PROGRAM MAIN

VAR
	fbSafetyX : fb_safety;
	fbSafetyY : fb_safety;
	fbSystemBufferX : fb_StatusBuffer;
	fbSystemBufferY : fb_StatusBuffer;
	fbMovementControllerX : fb_MovementController;
	fbMovementControllerY : fb_MovementController;
	fbBiaxialCoordinator : fb_BiaxialCoordinator;
	fbStatusPublisherX : fb_AxisStatusPublisher;
	fbStatusPublisherY : fb_AxisStatusPublisher;
	
	// DUTs import
	stMoveCommandX : ST_MoveCommand;
	stMoveCommandY : ST_MoveCommand;

	stSystemStatusX : ST_SystemStatus;
	stSystemStatusY : ST_SystemStatus;

	stSettingsX : ST_Settings;
	stSettingsY : ST_Settings;

	// IO Links
    nRawTenzoX AT %I* : DINT;
	nRawTenzoY AT %I* : DINT;

	nEndStopLx AT %I* : BOOL;
	nEndStopHx AT %I* : BOOL;

	nEndStopLy AT %I* : BOOL;
	nEndStopHy AT %I* : BOOL;

	// Normalized physical limits: TRUE means that the switch is pressed.
	bEndStopLxActive : BOOL;
	bEndStopHxActive : BOOL;
	bEndStopLyActive : BOOL;
	bEndStopHyActive : BOOL;

	// PLC-owned synchronized start request
	bStartBiaxialTest : BOOL; // ADS one-shot after both axis commands are prepared

	// Persistent-axis checkpoint diagnostics. A successful checkpoint creates
	// an up-to-date Port_851.bootdata file before controller power is removed.
	bPersistentPositionSaved : BOOL;
	bPersistentPositionSaveBusy : BOOL;
	bPersistentPositionSaveError : BOOL;
	nPersistentPositionSaveErrorID : UDINT;
	nPersistentPositionCheckpointCounter : UDINT;

	fbWritePersistentData : FB_WritePersistentData;
	fbPersistentPositionSettle : TON;
	ftPowerRequestX : F_TRIG;
	ftPowerRequestY : F_TRIG;
	rtPersistentValidX : R_TRIG;
	rtPersistentValidY : R_TRIG;
	bPersistentInitialCheckpoint : BOOL := TRUE;
	bPersistentCheckpointPending : BOOL;
	bPersistentCheckpointInFlight : BOOL;
	bPersistentCheckpointStart : BOOL;
	bPersistentSafeToWrite : BOOL;
	nPersistentCheckpointRequestGeneration : UDINT;
	nPersistentCheckpointStartedGeneration : UDINT;
	nPersistentCheckpointCompletedGeneration : UDINT;
	fCheckpointPositionX : LREAL;
	fCheckpointPositionY : LREAL;
	bCheckpointValidX : BOOL;
	bCheckpointValidY : BOOL;

END_VAR

VAR_TEMP
	bBiaxialAxesReady : BOOL;
	bBiaxialCommonAbortRequest : BOOL;
	bRestoreReferenceX : BOOL;
	bRestoreReferenceY : BOOL;
END_VAR

////////////////////////////////
//////////   safety   //////////
////////////////////////////////

// Refresh NC status before making any safety or motion decision
GVL_Axis.xAxis.ReadStatus();
GVL_Axis.yAxis.ReadStatus();

// Requesting a physical home deliberately invalidates the old retained
// coordinate. Only a successfully referenced axis will make it valid again.
IF stMoveCommandX.bHome THEN
	GVL_Persistent.bLastPositionValidX := FALSE;
END_IF
IF stMoveCommandY.bHome THEN
	GVL_Persistent.bLastPositionValidY := FALSE;
END_IF

// On the first powered scan after a PLC/NC restart, statically restore each
// incremental axis to its last persistent coordinate. MC_Direct performs no
// motor movement. A normal reference-cam home always takes priority.
bRestoreReferenceX :=
	GVL_Persistent.bLastPositionValidX AND
	NOT GVL_Axis.xAxis.Status.Homed AND
	NOT fbSafetyX.bReferenceRestoreDone;
bRestoreReferenceY :=
	GVL_Persistent.bLastPositionValidY AND
	NOT GVL_Axis.yAxis.Status.Homed AND
	NOT fbSafetyY.bReferenceRestoreDone;

// Normalize the active-low physical switches
bEndStopLxActive := NOT nEndStopLx;
bEndStopHxActive := NOT nEndStopHx;
bEndStopLyActive := NOT nEndStopLy;
bEndStopHyActive := NOT nEndStopHy;

fbSafetyX(
    stAxis := GVL_Axis.xAxis,
    bPower := stMoveCommandX.bPower,
    bReset := stMoveCommandX.bReset,
    bHalt := stMoveCommandX.bHalt OR fbMovementControllerX.stateHalt,
    bHome := stMoveCommandX.bHome,
	bRestoreReference := bRestoreReferenceX,
	fRestoreReferencePosition := GVL_Persistent.fLastPositionX,
    bEndStopL := bEndStopLxActive,
	bEndStopH := bEndStopHxActive,
	bExternalBusy := fbMovementControllerX.bBusy OR stSystemStatusX.bTarWorking
);

fbSafetyY(
    stAxis := GVL_Axis.yAxis,
    bPower := stMoveCommandY.bPower,
    bReset := stMoveCommandY.bReset,
    bHalt := stMoveCommandY.bHalt OR fbMovementControllerY.stateHalt,
    bHome := stMoveCommandY.bHome,
	bRestoreReference := bRestoreReferenceY,
	fRestoreReferencePosition := GVL_Persistent.fLastPositionY,
    bEndStopL := bEndStopLyActive,
	bEndStopH := bEndStopHyActive,
	bExternalBusy := fbMovementControllerY.bBusy OR stSystemStatusY.bTarWorking
);

////////////////////////////////
////////// Update data /////////
////////////////////////////////

fbSystemBufferX(
	stSystemStatus:= stSystemStatusX,
	bBlockTar:= fbMovementControllerX.bBusy OR fbSafetyX.bHoming OR
		NOT fbSafetyX.bHomed,
	nRawTenzo:= -nRawTenzoX,
	fTenzoCons:=stSettingsX.fTenzoCons,
	fTenzoOffset:= stSettingsX.fTenzoOffset,
	bStartTar:= stMoveCommandX.bStartTar,
	fActPosition:= GVL_Axis.xAxis.NcToPlc.ActPos);
	
fbSystemBufferY(
	stSystemStatus:= stSystemStatusY,
	bBlockTar:= fbMovementControllerY.bBusy OR fbSafetyY.bHoming OR
		NOT fbSafetyY.bHomed,
	nRawTenzo:= nRawTenzoY,
	fTenzoCons:=stSettingsY.fTenzoCons,
	fTenzoOffset:= stSettingsY.fTenzoOffset,
	bStartTar:= stMoveCommandY.bStartTar,
	fActPosition:= GVL_Axis.yAxis.NcToPlc.ActPos);

/////////////////////////////////////
////////// Main Move Logic //////////
/////////////////////////////////////

// A shared request starts both axes in one PLC scan. Single-axis tests keep
// using their individual bExecute fields and never enable synchronization.
bBiaxialAxesReady :=
	NOT fbMovementControllerX.bBusy AND
	NOT fbMovementControllerY.bBusy AND
	NOT fbMovementControllerX.bError AND
	NOT fbMovementControllerY.bError AND
	NOT fbSafetyX.bError AND NOT fbSafetyY.bError AND
	NOT fbSafetyX.bHoming AND NOT fbSafetyY.bHoming AND
	fbSafetyX.bHomed AND fbSafetyY.bHomed AND
	NOT stSystemStatusX.bTarWorking AND
	NOT stSystemStatusY.bTarWorking AND
	fbSafetyX.bPowerStatus AND fbSafetyY.bPowerStatus;

// Ignore ProtectiveStop when it was produced by the controller's own
// controlled halt. Operator, end-stop and independent safety stops abort both
// axes; an overforce relief request aborts only the synchronized peer.
bBiaxialCommonAbortRequest :=
	fbMovementControllerX.bError OR fbMovementControllerY.bError OR
	fbSafetyX.bError OR fbSafetyY.bError OR
	(fbSafetyX.bProtectiveStop AND
	 NOT fbMovementControllerX.stateHalt) OR
	(fbSafetyY.bProtectiveStop AND
	 NOT fbMovementControllerY.stateHalt) OR
	(bEndStopLxActive AND GVL_Axis.xAxis.Status.NegativeDirection) OR
	(bEndStopHxActive AND GVL_Axis.xAxis.Status.PositiveDirection) OR
	(bEndStopLyActive AND GVL_Axis.yAxis.Status.NegativeDirection) OR
	(bEndStopHyActive AND GVL_Axis.yAxis.Status.PositiveDirection) OR
	stMoveCommandX.bHalt OR stMoveCommandY.bHalt;

fbBiaxialCoordinator(
	bStartRequest := bStartBiaxialTest,
	bResetRequest := stMoveCommandX.bReset OR stMoveCommandY.bReset,
	bAxesReady := bBiaxialAxesReady,
	bCommonAbortRequest := bBiaxialCommonAbortRequest,
	bBusyX := fbMovementControllerX.bBusy,
	bBusyY := fbMovementControllerY.bBusy,
	bSavedPositionValidX := fbMovementControllerX.bSavedPositionValid,
	bSavedPositionValidY := fbMovementControllerY.bSavedPositionValid,
	nSyncPointX := fbMovementControllerX.nSyncPoint,
	nSyncPointY := fbMovementControllerY.nSyncPoint,
	nSyncCycleX := fbMovementControllerX.nSyncCycle,
	nSyncCycleY := fbMovementControllerY.nSyncCycle,
	bPeerAbortRequestX := fbMovementControllerX.bPeerAbortRequest,
	bPeerAbortRequestY := fbMovementControllerY.bPeerAbortRequest,
	stCommandX := stMoveCommandX,
	stCommandY := stMoveCommandY);

IF bStartBiaxialTest THEN
	bStartBiaxialTest := FALSE;
END_IF

IF fbBiaxialCoordinator.bStartBoth THEN
	stMoveCommandX.bExecute := TRUE;
	stMoveCommandY.bExecute := TRUE;
END_IF

fbMovementControllerX(
	Axis := GVL_Axis.xAxis,
	stMoveCommand := stMoveCommandX,
	stSettings := stSettingsX,
	fActPosition := GVL_Axis.xAxis.NcToPlc.ActPos,
    bPowerState := fbSafetyX.bPowerStatus,
	bHaltDone := fbSafetyX.bHaltDone,
	bAxisStopped := fbSafetyX.bStopped,
	bSafetyError := fbSafetyX.bError,
	bProtectiveStop := fbSafetyX.bProtectiveStop,
	bExternalBusy := fbSafetyX.bHoming OR
		NOT fbSafetyX.bHomed OR stSystemStatusX.bTarWorking,
	bReferenceValid := fbSafetyX.bHomed,
	bInvalidateSavedPosition := stMoveCommandX.bHome,
	bSyncEnabled := fbBiaxialCoordinator.bSyncActive,
	bSyncRelease := fbBiaxialCoordinator.bSyncRelease,
	bSyncAbort := fbBiaxialCoordinator.bAbortX,
	bSyncSingleComplete := fbBiaxialCoordinator.bSingleCompleteX,
    fForce := stSystemStatusX.fTenzoBuffer[stSystemStatusX.nBufferHead]);

fbMovementControllerY(
	Axis := GVL_Axis.yAxis,
	stMoveCommand := stMoveCommandY,
	stSettings := stSettingsY,
	fActPosition := GVL_Axis.yAxis.NcToPlc.ActPos,
    bPowerState := fbSafetyY.bPowerStatus,
	bHaltDone := fbSafetyY.bHaltDone,
	bAxisStopped := fbSafetyY.bStopped,
	bSafetyError := fbSafetyY.bError,
	bProtectiveStop := fbSafetyY.bProtectiveStop,
	bExternalBusy := fbSafetyY.bHoming OR
		NOT fbSafetyY.bHomed OR stSystemStatusY.bTarWorking,
	bReferenceValid := fbSafetyY.bHomed,
	bInvalidateSavedPosition := stMoveCommandY.bHome,
	bSyncEnabled := fbBiaxialCoordinator.bSyncActive,
	bSyncRelease := fbBiaxialCoordinator.bSyncRelease,
	bSyncAbort := fbBiaxialCoordinator.bAbortY,
	bSyncSingleComplete := fbBiaxialCoordinator.bSingleCompleteY,
	fForce := stSystemStatusY.fTenzoBuffer[stSystemStatusY.nBufferHead]);

///////////////////////////////////////////////////
////// ADS status contract for each axis //////////
///////////////////////////////////////////////////

fbStatusPublisherX(
	fActPosition := GVL_Axis.xAxis.NcToPlc.ActPos,
	bPowerStatus := fbSafetyX.bPowerStatus,
	bHoming := fbSafetyX.bHoming,
	bHomed := fbSafetyX.bHomed,
	bStopped := fbSafetyX.bStopped,
	bProtectiveStop := fbSafetyX.bProtectiveStop,
	bControllerHalt := fbMovementControllerX.stateHalt,
	bSafetyError := fbSafetyX.bError,
	nSafetyErrorCode := fbSafetyX.nErrorCode,
	nSafetyAxisErrorID := fbSafetyX.nAxisErrorID,
	bMovementBusy := fbMovementControllerX.bBusy,
	bMovementError := fbMovementControllerX.bError,
	nMovementStatus := fbMovementControllerX.nSystemStatus,
	nMovementErrorCode := fbMovementControllerX.nErrorCode,
	nMovementAxisErrorID := fbMovementControllerX.nAxisErrorID,
	nOperationCounter := fbMovementControllerX.nOperationCounter,
	bSavedPositionValid := fbMovementControllerX.bSavedPositionValid,
	bStartError := fbBiaxialCoordinator.bStartError,
	nStartErrorCode := fbBiaxialCoordinator.nStartErrorCode,
	stSystemStatus := stSystemStatusX);

fbStatusPublisherY(
	fActPosition := GVL_Axis.yAxis.NcToPlc.ActPos,
	bPowerStatus := fbSafetyY.bPowerStatus,
	bHoming := fbSafetyY.bHoming,
	bHomed := fbSafetyY.bHomed,
	bStopped := fbSafetyY.bStopped,
	bProtectiveStop := fbSafetyY.bProtectiveStop,
	bControllerHalt := fbMovementControllerY.stateHalt,
	bSafetyError := fbSafetyY.bError,
	nSafetyErrorCode := fbSafetyY.nErrorCode,
	nSafetyAxisErrorID := fbSafetyY.nAxisErrorID,
	bMovementBusy := fbMovementControllerY.bBusy,
	bMovementError := fbMovementControllerY.bError,
	nMovementStatus := fbMovementControllerY.nSystemStatus,
	nMovementErrorCode := fbMovementControllerY.nErrorCode,
	nMovementAxisErrorID := fbMovementControllerY.nAxisErrorID,
	nOperationCounter := fbMovementControllerY.nOperationCounter,
	bSavedPositionValid := fbMovementControllerY.bSavedPositionValid,
	bStartError := fbBiaxialCoordinator.bStartError,
	nStartErrorCode := fbBiaxialCoordinator.nStartErrorCode,
	stSystemStatus := stSystemStatusY);

// Track the last valid coordinate continuously in persistent PLC memory.
// Values are never replaced while an axis is unreferenced, homing, or in an
// NC error, so startup cannot accidentally retain the raw zero coordinate.
IF fbSafetyX.bHomed AND NOT fbSafetyX.bHoming AND
	NOT GVL_Axis.xAxis.Status.Error AND
	(GVL_Axis.xAxis.NcToPlc.ActPos =
		GVL_Axis.xAxis.NcToPlc.ActPos) AND
	ABS(GVL_Axis.xAxis.NcToPlc.ActPos) < 1.0E300 THEN
	GVL_Persistent.fLastPositionX :=
		GVL_Axis.xAxis.NcToPlc.ActPos;
	GVL_Persistent.bLastPositionValidX := TRUE;
END_IF

IF fbSafetyY.bHomed AND NOT fbSafetyY.bHoming AND
	NOT GVL_Axis.yAxis.Status.Error AND
	(GVL_Axis.yAxis.NcToPlc.ActPos =
		GVL_Axis.yAxis.NcToPlc.ActPos) AND
	ABS(GVL_Axis.yAxis.NcToPlc.ActPos) < 1.0E300 THEN
	GVL_Persistent.fLastPositionY :=
		GVL_Axis.yAxis.NcToPlc.ActPos;
	GVL_Persistent.bLastPositionValidY := TRUE;
END_IF

///////////////////////////////////////////////////
//// Persistent coordinate disk checkpoint ///////
///////////////////////////////////////////////////

// PERSISTENT values in RAM are normally copied to Port_851.bootdata only on
// an orderly TwinCAT stop. Create a checkpoint after a normal home and when
// the operator removes commanded motor power so a later hard power-off does
// not fall back to an older coordinate. Never write continuously while the
// axes move; that would both save an unsafe intermediate coordinate and wear
// the controller's flash storage.
ftPowerRequestX(CLK := stMoveCommandX.bPower);
ftPowerRequestY(CLK := stMoveCommandY.bPower);
rtPersistentValidX(CLK := GVL_Persistent.bLastPositionValidX);
rtPersistentValidY(CLK := GVL_Persistent.bLastPositionValidY);

IF bPersistentInitialCheckpoint OR ftPowerRequestX.Q OR
	ftPowerRequestY.Q OR rtPersistentValidX.Q OR
	rtPersistentValidY.Q THEN
	bPersistentCheckpointPending := TRUE;
	nPersistentCheckpointRequestGeneration :=
		nPersistentCheckpointRequestGeneration + 1;
	bPersistentPositionSaved := FALSE;
	bPersistentPositionSaveError := FALSE;
	nPersistentPositionSaveErrorID := 0;
	bPersistentInitialCheckpoint := FALSE;
END_IF

// Mark the public diagnostic false as soon as a referenced coordinate moves
// away from the last successfully written snapshot. A new disk write remains
// intentionally tied to home/power-off rather than every test endpoint.
IF bPersistentPositionSaved AND (
	(GVL_Persistent.bLastPositionValidX <>
		bCheckpointValidX) OR
	(GVL_Persistent.bLastPositionValidY <>
		bCheckpointValidY) OR
	(GVL_Persistent.bLastPositionValidX AND
		ABS(GVL_Persistent.fLastPositionX -
			fCheckpointPositionX) > 0.001) OR
	(GVL_Persistent.bLastPositionValidY AND
		ABS(GVL_Persistent.fLastPositionY -
			fCheckpointPositionY) > 0.001)) THEN
	bPersistentPositionSaved := FALSE;
END_IF

// Wait for a stable non-moving state before writing. An already loaded
// persistent coordinate may be checkpointed while its axis is unpowered; if
// powered, the NC axis must be referenced, stopped and error-free.
bPersistentSafeToWrite :=
	(GVL_Persistent.bLastPositionValidX OR
		GVL_Persistent.bLastPositionValidY) AND
	NOT fbMovementControllerX.bBusy AND
	NOT fbMovementControllerY.bBusy AND
	NOT fbSafetyX.bHoming AND NOT fbSafetyY.bHoming AND
	NOT stSystemStatusX.bTarWorking AND
	NOT stSystemStatusY.bTarWorking AND
	(NOT fbSafetyX.bPowerStatus OR
		(fbSafetyX.bHomed AND fbSafetyX.bStopped AND
			NOT GVL_Axis.xAxis.Status.Error)) AND
	(NOT fbSafetyY.bPowerStatus OR
		(fbSafetyY.bHomed AND fbSafetyY.bStopped AND
			NOT GVL_Axis.yAxis.Status.Error));

fbPersistentPositionSettle(
	IN := bPersistentCheckpointPending AND
		NOT bPersistentCheckpointInFlight AND
		bPersistentSafeToWrite,
	PT := T#1S);

bPersistentCheckpointStart :=
	fbPersistentPositionSettle.Q AND
	NOT fbWritePersistentData.BUSY AND
	NOT bPersistentCheckpointInFlight;

fbWritePersistentData(
	NETID := '',
	PORT := TwinCAT_SystemInfoVarList._AppInfo.AdsPort,
	START := bPersistentCheckpointStart,
	TMOUT := T#5S,
	MODE := SPDM_VAR_BOOST);

IF bPersistentCheckpointStart THEN
	bPersistentCheckpointInFlight := TRUE;
	nPersistentCheckpointStartedGeneration :=
		nPersistentCheckpointRequestGeneration;
	fCheckpointPositionX := GVL_Persistent.fLastPositionX;
	fCheckpointPositionY := GVL_Persistent.fLastPositionY;
	bCheckpointValidX := GVL_Persistent.bLastPositionValidX;
	bCheckpointValidY := GVL_Persistent.bLastPositionValidY;
ELSIF bPersistentCheckpointInFlight AND
	NOT fbWritePersistentData.BUSY THEN
	bPersistentCheckpointInFlight := FALSE;
	nPersistentCheckpointCompletedGeneration :=
		nPersistentCheckpointStartedGeneration;
	bPersistentCheckpointPending :=
		nPersistentCheckpointCompletedGeneration <>
		nPersistentCheckpointRequestGeneration;
	IF fbWritePersistentData.ERR THEN
		bPersistentPositionSaved := FALSE;
		bPersistentPositionSaveError := TRUE;
		nPersistentPositionSaveErrorID :=
			fbWritePersistentData.ERRID;
	ELSE
		bPersistentPositionSaved := TRUE;
		bPersistentPositionSaveError := FALSE;
		nPersistentPositionSaveErrorID := 0;
		nPersistentPositionCheckpointCounter :=
			nPersistentPositionCheckpointCounter + 1;
	END_IF
END_IF

bPersistentPositionSaveBusy :=
	bPersistentCheckpointPending OR
	bPersistentCheckpointInFlight OR
	fbWritePersistentData.BUSY;

// Home and reset are one-shot commands
stMoveCommandX.bHome := FALSE;
stMoveCommandY.bHome := FALSE;
stMoveCommandX.bReset := FALSE;
stMoveCommandY.bReset := FALSE;
stMoveCommandX.bSavePosition := FALSE;
stMoveCommandY.bSavePosition := FALSE;
stMoveCommandX.bRestorePosition := FALSE;
stMoveCommandY.bRestorePosition := FALSE;

END_PROGRAM

(* stored: Version 1.1.0.1, ProductVersion 3.1.4024.15
   POU MAIN: Id {6bc6223d-2cd4-47db-ac9d-d10a27a83f14}, SpecialFunc None *)
